TYPE SC_BUSY_BeltConveyors :
(
	eBusySCStart := 0,
	eStartEntranceConveyor,
	eStartUpwardsConveyor,
	eExecutePalletizer,
	eSignalError
)UINT;
END_TYPE

(* stored: Version 1.1.0.1, ProductVersion 3.1.4024.0
   DUT SC_BUSY_BeltConveyors: Id {d8dd3c01-09dc-42da-a6f4-d0bfc8d0fd61} *)
